FUNCTION_BLOCK EnableDisbableTask IMPLEMENTS I_Task, I_Cyclic, I_Object, I_Abortable
VAR
	mcPower : Tc2_MC2.MC_Power;
	_Axis : REFERENCE TO Tc2_MC2.AXIS_REF;
	_InhibitPos : BOOL := FALSE;
	_InhibitNeg : BOOL := FALSE;
END_VAR

{analysis -2}

METHOD Abort : HRESULT
mcPower.Enable := FALSE;
mcPower.Enable_Negative := FALSE;
mcPower.Enable_Positive := FALSE;
END_METHOD

PROPERTY AxisRef : reference to Axis_Ref
GET // PUBLIC
AxisRef REF= _Axis;
END_GET
SET
_Axis REF= AxisRef;
END_SET
END_PROPERTY

PROPERTY Busy : BOOL
GET
Busy := mcPower.Busy;
END_GET
END_PROPERTY

METHOD Cycle : HRESULT
VAR_INPUT
END_VAR
mcPower(Axis := _Axis);
END_METHOD

METHOD Disable : HRESULT
VAR_INPUT

END_VAR
mcPower.Enable := FALSE;
END_METHOD

PROPERTY Done : BOOL
GET
Done := NOT mcPower.Busy;
END_GET
END_PROPERTY

METHOD Enable : HRESULT
VAR_INPUT
END_VAR
mcPower.Enable := TRUE;
mcPower.Enable_Negative := NOT _InhibitNeg;
mcPower.Enable_Positive := NOT _InhibitPos;
END_METHOD

PROPERTY Error : BOOL
GET
Error := mcPower.Error;
END_GET
END_PROPERTY

PROPERTY InhibitNegative : BOOL
GET
InhibitNegative := _InhibitNeg;
END_GET
SET
_InhibitNeg := InhibitNegative;
END_SET
END_PROPERTY

PROPERTY InhibitPositive : BOOL
GET
InhibitPositive := _InhibitPos;
END_GET
SET
_InhibitPos := InhibitPositive;
END_SET
END_PROPERTY

METHOD RegisterWithParent
VAR_INPUT
	Runner	: I_HostObjects;
END_VAR
Runner.RegisterAbortable(THIS^);
Runner.RegisterCyclic(THIS^);
Runner.RegisterTask(THIS^);
END_METHOD

END_FUNCTION_BLOCK

(* stored: Version 1.1.0.1
   POU EnableDisbableTask: Id {9020922a-7816-4155-9202-ac5854f794ea}, SpecialFunc None
   Method Abort: Id {93bd9e75-34cf-4a99-8cdf-c273723a870d}
   Property AxisRef: Id {4f69ca7b-ca74-4b65-bdce-7eb1296f6878}
   Get Get: Id {ac8e833e-ec0c-44ce-9087-839c459ac896}
   Set Set: Id {244ac82c-e273-4291-b98b-549fb47607b8}
   Property Busy: Id {c798d0d0-97d0-4d53-b519-da00d5dccc4f}
   Get Get: Id {c431141b-efc9-4560-8025-c7c0a08af50a}
   Method Cycle: Id {c1cf1940-bcdc-4ac4-844e-317c1f14fe0e}
   Method Disable: Id {0a54e8c6-7456-4747-8eeb-b97b9078e709}
   Property Done: Id {006aa190-9c68-4a73-bf0c-8a7f7aaf57ff}
   Get Get: Id {3155aba1-6f22-460f-ac4b-c62ed8476ecf}
   Method Enable: Id {afe5d65c-4532-4d19-b244-08cfed3445ed}
   Property Error: Id {518ce1d0-c80e-419e-af03-bf594c64bec9}
   Get Get: Id {f9e74dcb-6dbd-485e-b208-5c6b8f34d064}
   Property InhibitNegative: Id {dc288d3e-02f1-4405-a301-d619e78f06f3}
   Get Get: Id {0424fba8-b630-4cde-9947-0bd6ec5b0728}
   Set Set: Id {acc383d4-6fb0-4c6a-91e8-44a029dd8dfe}
   Property InhibitPositive: Id {610d9724-51d9-4637-ac8e-5c718072673e}
   Get Get: Id {726bca85-749b-4131-8cb6-fe4c20afdfd9}
   Set Set: Id {b3374342-2590-4bb5-9407-5b6a52700a4b}
   Method RegisterWithParent: Id {a33ff5bc-abb9-465a-9880-0802eec356db} *)
